# EPICS autosave request: 3-0/GalilSup/Db/galil_analog_in.req
$(P)$(R)_MON.DESC
